// Counts how many tests are inside their body at the same moment.
//
// A test cannot observe this about another test - it is handed nothing but its own
// assertion handle, which is the founding constraint working as intended.
//
// So tests report in and out of a shared witness instead, and the contract becomes
// one number: MaxConcurrent must never exceed 1.
FUNCTION_BLOCK ConcurrencyWitness
VAR
	_Active		   : DINT;
	_MaxConcurrent : DINT;
	_TotalEntries  : DINT;
END_VAR

// A test body has started. Called on its FIRST scan only.
METHOD Enter
_Active		  := _Active + 1;
_TotalEntries := _TotalEntries + 1;

IF _Active > _MaxConcurrent THEN
	_MaxConcurrent := _Active;
END_IF
END_METHOD

// A test body has finished. Called on its LAST scan only.
METHOD Leave
_Active := _Active - 1;
END_METHOD

// The most tests ever inside a body at once. Must be 1: tests share the scan and
// usually share fixtures, so predictable and slow beats fast and flaky.
PROPERTY MaxConcurrent : DINT
GET
MaxConcurrent := _MaxConcurrent;
END_GET
END_PROPERTY

METHOD Reset
_Active		   := 0;
_MaxConcurrent := 0;
_TotalEntries  := 0;
END_METHOD

// How many bodies started. Proves every test really ran, so a MaxConcurrent of 1
// cannot be achieved by nothing running at all.
PROPERTY TotalEntries : DINT
GET
TotalEntries := _TotalEntries;
END_GET
END_PROPERTY

END_FUNCTION_BLOCK

(* stored: Version 1.1.0.1, ProductVersion 3.1.4026.18
   POU ConcurrencyWitness: Id {ca0af444-af45-44d7-a1a9-f6350d96227d}, SpecialFunc None
   Method Enter: Id {5cfb1517-20d5-4773-8606-e602988522bd}
   Method Leave: Id {08f97010-fe51-484a-b857-a68bad225dda}
   Property MaxConcurrent: Id {e7c61d99-c4e2-4932-ba6b-304b230937c6}
   Get Get: Id {6cac1f46-a67c-4608-89bf-0d1f9671d8e2}
   Method Reset: Id {4412c1dc-590d-4427-ac9d-401dff8e854f}
   Property TotalEntries: Id {f22b6435-2944-4456-ab93-2435271813ba}
   Get Get: Id {a8027ec6-9d5d-4d25-954c-9a2c4740c9f1} *)
